(* CODESYS project 2.project

Project tree, tasks and I/O mapping:
  Device : CODESYS Control Win V3, 3S - Smart Software Solutions GmbH, order no. 305021, version 3.5.11.30
    application Application
      libraries: Standard, * (System)
      task MainTask (cyclic, interval t#20ms, priority 1) calls PLC_PRG
      program PLC_PRG [LD]
*)

// Device/Application/PLC_PRG
PROGRAM PLC_PRG
VAR 
	A: BOOL;
	B: BOOL;
	C: BOOL;
	OUT: BOOL;
	
END_VAR

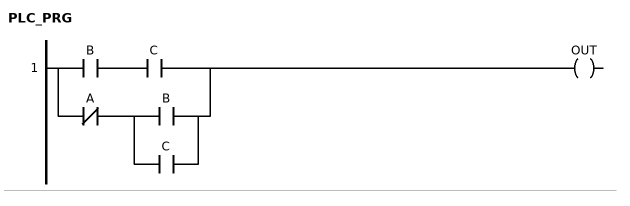
// NETWORK 1
OUT := B AND C OR NOT A AND (B OR C);

END_PROGRAM
